(* CODESYS project snapsignal_board
   CompiledLibraryCompatibilityVersion: CODESYS V3.5 SP16 Patch 3

Project tree, tasks and I/O mapping:
  Device : TX707/TX707HB-P3CV01, Turck, order no. 100002030/100007473, version 3.5.16.30
    application Application
      libraries: Standard, 3.5.18.0 (System); VisuElemBase, * (System); CmpBitmapPool, * (System); VisuDialogs, * (System)
      task ENIPScannerIOTask (cyclic, interval t#10ms, priority 0) calls EtherNet_IP_Scanner.IOCycle
      task ENIPScannerServiceTask (cyclic, interval t#20ms, priority 30) calls EtherNet_IP_Scanner.ServiceCycle
      task MainTask (cyclic, interval 10 ms, priority 1) calls POU
      task VISU_TASK (cyclic, interval 100 ms, priority 31) calls VisuElems.Visu_Prg
      program CURRENT [ST]
      visualisation Current_screen
      image pool ImagePool
      visualisation Linear_pos_screen
      program LPOS [ST]
      visualisation Main_screen
      program POU [ST]
      program VIBRATION [ST]
      visualisation Vibration_temp_screen
    Ethernet : Ethernet, CODESYS, version 4.2.0.0
        settings: IPAddress = [192,168,15,15]; SubnetMask = [255,255,255,0]; GatewayAddress = [0,0,0,0]; MACAddress = [16#00,16#07,16#46,16#25,16#94,16#63]; NetworkInterfaceName = 'br0'; NetworkInterfaceName = "br0"; SaveCommunicationSettings = FALSE; IPAddress = [192,168,0,2]; SubnetMask = [255,255,255,0]; GatewayAddress = [0,0,0,0]
      EtherNet_IP_Scanner : EtherNet/IP Scanner, CODESYS, order no. 1, version 4.5.1.0
  libraries: VisuSymbols, 4.5.0.0 (System)
  5ce3da45-db07-42e7-a21c-a00fff4ed8f6|C:\Users\juszuf.arsunkaev\Desktop\linear.jpg
  5ce3da45-db07-42e7-a21c-a00fff4ed8f6|C:\Users\juszuf.arsunkaev\Downloads\linear.jpeg
  5ce3da45-db07-42e7-a21c-a00fff4ed8f6|C:\Users\juszuf.arsunkaev\Downloads\Q2XKLAFAIR-Q_812837_sideD.psd - 319 x 319.png
  5ce3da45-db07-42e7-a21c-a00fff4ed8f6|C:\Users\juszuf.arsunkaev\Downloads\qm30vt2-212030-front.psd - 319 x 319.png
  5ce3da45-db07-42e7-a21c-a00fff4ed8f6|C:\Users\juszuf.arsunkaev\Downloads\turck_logo_download.jpg
  GlobalImagePool
  text list GlobalTextList
*)

// Device/Application/POU
PROGRAM POU
VAR
	 g_ActiveDevice : INT := 3;
	 PageIndex :INT;
	 SwitchTimer: TON;
	 SwitchDelay : TIME := T#1000MS;
END_VAR


// Timer set to prevent PageIndex incrementing/decrementing too fast when buttons are pressed
SwitchTimer(IN := (display_41_button = 1 OR display_41_button = 2), PT := SwitchDelay);

// Making sure POUs don't run simultaneously
CASE g_ActiveDevice OF
    0: CURRENT();
    1: VIBRATION();
    2: LPOS();
    3: ; // No POU runs when on home screen
END_CASE

IF CurrentVisu = 'Current_screen' THEN
    g_ActiveDevice := 0;
ELSIF CurrentVisu = 'Vibration_temp_screen' THEN
    g_ActiveDevice := 1;
ELSIF CurrentVisu = 'Linear_pos_screen' THEN
    g_ActiveDevice := 2;
ELSIF CurrentVisu = 'Main_screen' THEN
    g_ActiveDevice := 3;
    display_41_colour := 1;
    display_40_colour := 1;
    display_40 := 0;
    display_41 := 0;
END_IF

// Increment/Decrement PageIndex when display_41_button is pressed logic
IF SwitchTimer.Q THEN
    IF display_41_button = 2 THEN // Up button pressed
        PageIndex := PageIndex + 1;
		actuated_41_color := 5;
        IF PageIndex > 4 THEN
            PageIndex := 1; // Wrap around to the first page
        END_IF
    ELSIF display_41_button = 1 THEN // Down button pressed
        PageIndex := PageIndex - 1;
		actuated_41_color := 12;
        IF PageIndex < 1 THEN
            PageIndex := 4; // Wrap around to the last page
        END_IF
    END_IF
    // Reset the timer
    SwitchTimer(IN := FALSE);
END_IF


// Logic to switch the frame content based on PageIndex
CASE PageIndex OF
    1: CurrentVisu := 'Main_screen';
    2: CurrentVisu := 'Current_screen';
    3: CurrentVisu := 'Linear_pos_screen';
    4: CurrentVisu := 'Vibration_temp_screen';
END_CASE

END_PROGRAM

// Device/Application/CURRENT
PROGRAM CURRENT

VAR
	ct_value AT %IW156: WORD;
	display_41 AT %QW124: WORD;
	display_41_colour AT %QW125: WORD;
END_VAR

IF  CurrentVisu = 'Main_screen' THEN
			display_41 := 0;
			display_41_colour := 1;
			display_40 := 0;
			display_40_colour := 1;
		END_IF

IF CurrentVisu = 'Current_screen' THEN
    display_41 := TO_WORD(ct_value) * 10;
	//K50 display color changing logic based on ct_value
    IF ct_value >= 12 THEN
        display_41_colour := 7;
        IF ct_value >= 17 THEN
            display_41_colour := 0;
        END_IF
    ELSE 
        display_41_colour := 13;
    END_IF
END_IF

END_PROGRAM

// Device/Application/VIBRATION
PROGRAM VIBRATION
VAR
	vibration_z AT %IW158: WORD;
	vibration_x AT %IW159: WORD;
	rvib_z: REAL;
	rvib_x: REAL;
	display_41 AT %QW124: WORD;
	display_41_colour AT %QW125: WORD := 1;
	display_40 AT %QW126: WORD;
	display_40_colour AT %QW127: WORD:= 1;
	temperature_celsius: REAL;
	temperature_scaled: REAL;
END_VAR

rvib_z := TO_REAL(vibration_z) / 1000;
rvib_x := TO_REAL(vibration_x) / 1000;
temperature_scaled := TO_REAL(temperature)/100;
temperature_celsius := (temperature_scaled-32)*0.555;


display_41 := TO_WORD(rvib_z);
display_40 := TO_WORD(rvib_x);

//If user is on the main screen the display values are set to 0 for now
IF  CurrentVisu = 'Main_screen' THEN
			display_41 := 0;
			display_40 := 0;
		ELSIF CurrentVisu = 'Vibration_screen' THEN
    	display_41 := TO_WORD(ct_value) * 10;
		END_IF
		//K50 display color changing logic
		IF rvib_z>=3 THEN
			display_41_colour:=7;
			IF rvib_z>=8 THEN
				display_41_colour:=0;
			END_IF
			ELSE display_41_colour:=1;
		END_IF
	
		IF rvib_x>=3 THEN
			display_40_colour:=7;
			IF rvib_x>=8 THEN
				display_40_colour:=0;
			END_IF
		ELSE 
			display_40_colour:=1;
		END_IF

END_PROGRAM

// Device/Application/LPOS
PROGRAM LPOS
VAR
	position_mm : WORD;
END_VAR

//Added this because the process data ends in an awkward place on the sensor
IF linear_position < 235 THEN
	position_mm := 0;
	ELSIF linear_position > 17020 THEN
		position_mm := 100;
		ELSE position_mm := (linear_position - 235) * 100 / 17004;
END_IF

END_PROGRAM

// Device/Application/Current_screen
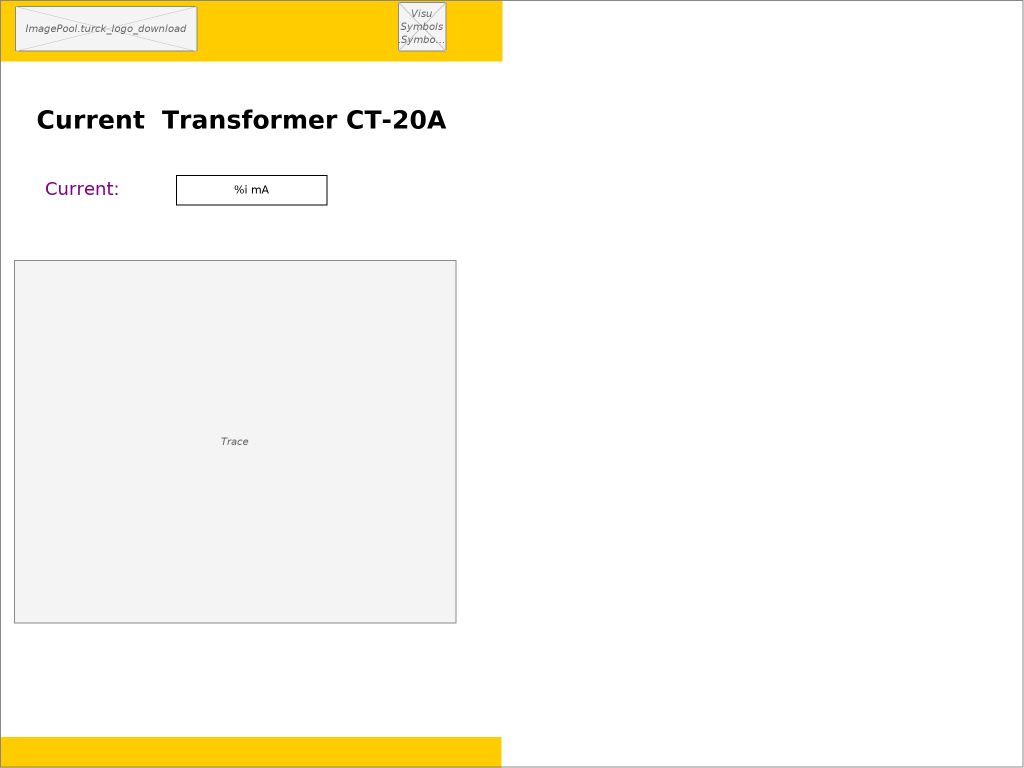
VISUALIZATION Current_screen  // 1024x768
    Trace (14,260 442x363)
    Label (-9,158 150x30)
    Label (-17,105 517x29), "Current Transformer CT-20A"
    Label (15,174 135x30), "Current:"
    Rectangle (176,175 151x30), "%i mA", text variable: CURRENT.display_41
    Rectangle (0,-2 502x63)
    Image (15,6 182x45), image: ImagePool.turck_logo_download
    Rectangle (-1,737 502x63)
    Image (398,2 48x49), image: VisuSymbols.Symbols.Home
        OnMouseClick: execute { POU.PageIndex:=1; }
END_VISUALIZATION

// Device/Application/Linear_pos_screen
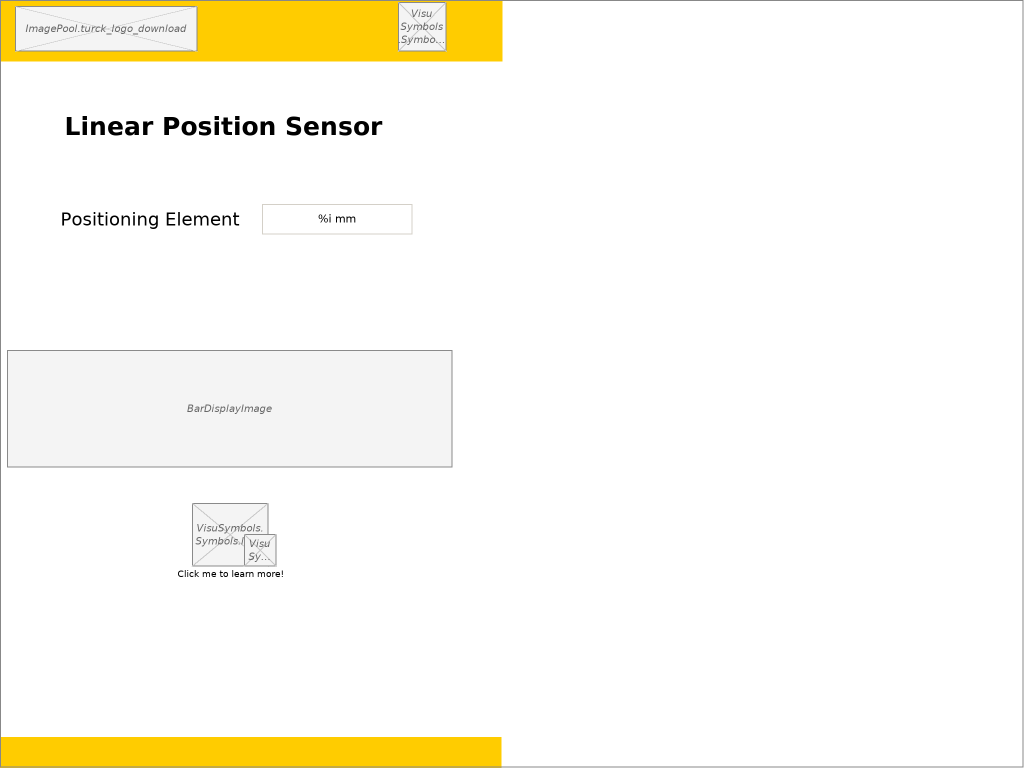
VISUALIZATION Linear_pos_screen  // 1024x768
    Label (32,111 392x30), "Linear Position Sensor"
    Rectangle (0,-2 502x63)
    Image (398,2 48x49), image: VisuSymbols.Symbols.Home
        OnMouseClick: execute { POU.PageIndex:=1; }
    Image (15,6 182x45), image: ImagePool.turck_logo_download
    Group (-1,737 502x63)
        Rectangle (0,0 502x63)
        Button (339,15 106x30), "Next"
            OnMouseClick:  Assign=Linear_pos_screen, Type=Assignment
        Button (34,15 106x30), "Back"
            OnMouseClick:  Assign=Vibration_temp_screen, Type=Assignment
    BarDisplayImage (7,350 445x117), value: LPOS.position_mm, style: BarDisplayImage-Gray, scale format: %.1f, scale 0..100
        p3451962224: ImagePool.linear0
    Textfield (262,204 150x30), "%i mm", text variable: LPOS.position_mm
    Label (7,196 286x47), "Positioning Element"
    Image (192,503 76x63), tooltip "The measuring principle of linear position sensors is based on RLC coupling between the positioning element and the sensor, whereby an output signal is provided proportional to the position of the positioning element. The rugged sensors are wear and tear-free, thanks to the contactless operating principle.", image: VisuSymbols.Symbols.light
    Label (156,559 150x30), "Click me to learn more!"
    Image (244,534 32x32), image: VisuSymbols.Symbols.ArrowQuarterLeftLeft
    Rectangle (-1,737 502x63)
END_VISUALIZATION

// Device/Application/Main_screen
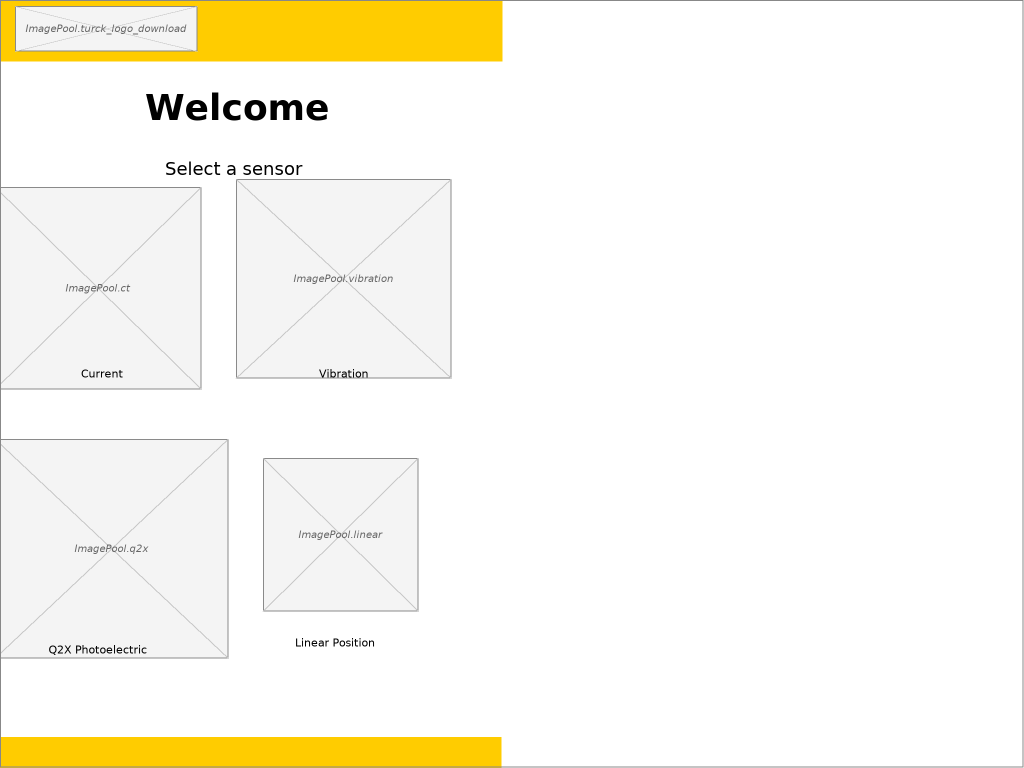
VISUALIZATION Main_screen  // 1024x768
    Label (126,71 223x73), "Welcome"
    Image (-5,187 206x202), image: ImagePool.ct
        OnMouseClick:  Assign=Current_screen, Type=Assignment
        OnMouseClick: execute { POU.PageIndex := 2; }
    Image (236,179 215x199), image: ImagePool.vibration
        OnMouseClick:  Assign=Vibration_temp_screen, Type=Assignment
        OnMouseClick: execute { POU.PageIndex := 4; }
    Image (-5,439 233x219), image: ImagePool.q2x
    Image (263,458 155x153), image: ImagePool.linear
        OnMouseClick:  Assign=Linear_pos_screen, Type=Assignment
        OnMouseClick: execute { POU.PageIndex := 3; }
    Rectangle (0,-2 502x63)
    Image (15,6 182x45), image: ImagePool.turck_logo_download
    Rectangle (-1,737 502x63)
    Label (40,154 388x30), "Select a sensor"
    Label (27,359 150x30), "Current"
    Label (269,359 150x30), "Vibration"
    Label (23,635 150x30), "Q2X Photoelectric"
    Label (260,628 150x30), "Linear Position"
END_VISUALIZATION

// Device/Application/Vibration_temp_screen
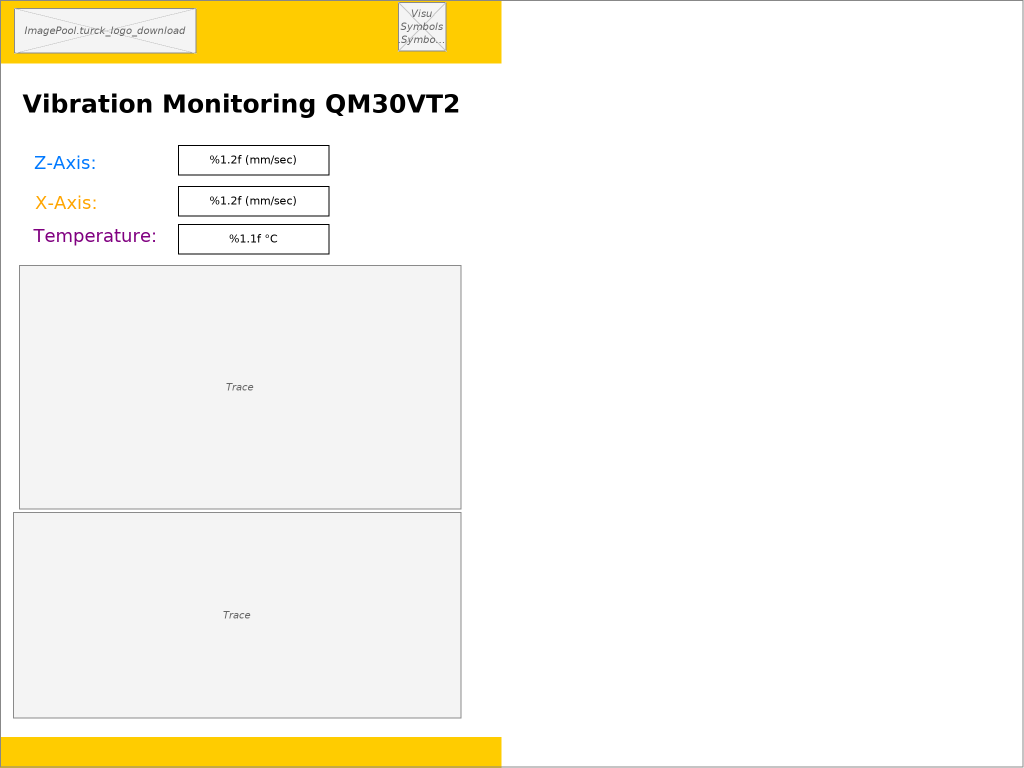
VISUALIZATION Vibration_temp_screen  // 1024x768
    Trace (19,265 442x244)
    Label (-7,148 150x30), "Z-Axis:"
    Label (-6,188 150x30), "X-Axis:"
    Rectangle (178,145 151x30), "%1.2f (mm/sec)", text variable: VIBRATION.rvib_z
    Rectangle (178,186 151x30), "%1.2f (mm/sec)", text variable: VIBRATION.rvib_x
    Label (-17,89 517x29), "Vibration Monitoring QM30VT2"
    Label (28,221 135x30), "Temperature:"
    Rectangle (178,224 151x30), "%1.1f °C", text variable: VIBRATION.temperature_celsius
    Trace (13,512 448x206)
    Rectangle (-1,0 502x63)
    Image (14,8 182x45), image: ImagePool.turck_logo_download
    Group (-2,739 502x63)
        Rectangle (0,0 502x63)
        Button (339,15 106x30), "Next"
            OnMouseClick:  Assign=Current_screen, Type=Assignment
        Button (34,15 106x30), "Back"
            OnMouseClick:  Assign=Linear_pos_screen, Type=Assignment
    Rectangle (-1,737 502x63)
    Image (398,2 48x49), image: VisuSymbols.Symbols.Home
        OnMouseClick: execute { POU.PageIndex:=1; }
END_VISUALIZATION
